TYPE "Component Check_ShW"
VERSION : 0.1
   STRUCT
      Trigger : Bool;
      Q_ID : "ComponentID_ShW";
      IDResult : Int;
      IDResult1 : Array[1..10] of Int;
      Completed : Bool;
   END_STRUCT;

END_TYPE

